(* PLC project Generated.project, CODESYS CODESYS V3.5 SP19 Patch 1 *)
(* stored: creationDateTime 2026-08-18T12:52:51.329350, modificationDateTime 2026-08-18T12:52:51.329350 *)

(* ═══════════════════════════════════════════════════════════════ 🚦 ST_SyncState — États et diagnostics de la synchronisation M1/M2 ═══════════════════════════════════════════════════════════════ *)
TYPE ST_SyncState : STRUCT
  DeltaPos_M : REAL;  (* 📊 Écart de position réel mesuré (m) *)
  SyncActive : BOOL;  (* ⚖️ Indicateur si surveillance active *)
  SyncWarn : BOOL;  (* ⚠️ LED d'alarme écart hors tolérance *)
  SyncDegradedStep1 : BOOL;  (* 🐢 Écart modéré actif : limitation forcée au Palier 1 *)
  Ready : BOOL;  (* 🟢 Bloc de synchro prêt *)
  Error : BOOL;  (* Alarme synchro active *)
  ErrorId : WORD;  (* ❌ Code défaut synchro *)
  FBState : E_State;  (* 🤖 État de l'automate interne (FB_WinchSync) — ex-"State", renommé pour éviter collision avec le sous-struct State *)
END_STRUCT;
END_TYPE

(* values of E_State: DISABLED: Enable faux, neutralisé; INIT: Démarrage / vérifs; READY: Prêt, attend ordre; BUSY: Action en cours; DONE: Action terminée; STOPPING: Décél rampe avant arrêt (StartStop=FALSE ou SafeStop=TRUE) *)

{attribute 'qualified_only'}
{attribute 'strict'}
TYPE E_State : (DISABLED := 0, INIT := 1, READY := 2, BUSY := 3, DONE := 4, STOPPING := 5);
END_TYPE
